# EPICS autosave request: support/areaDetector/1-4/iocBoot/iocAdsc/auto_settings.req
file "ADBase_settings.req", P=$(P),  R=det1:
file "adsc_settings.req",   P=$(P),  R=det1:
